TYPE (* An Array Data Type *)
  (* Standard: 61131-3 *)
  (* Version 0.0, 2003-12-06, JHC, Rockwell Automation *)
  (* Compiler header: package fb.rt.template; *)
  (* ASN.1 tag PRIVATE 8 *)
  Array : ARRAY [0..4] OF REAL := [1,2,3,4,5];
END_TYPE
